INTERFACE I_EnumeratorConnectionItem

END_INTERFACE

(* stored: Version 1.1.0.1, ProductVersion 3.1.4024.12
   Itf I_EnumeratorConnectionItem: Id {e091440f-74bb-44c5-bffa-19176a69207f} *)
